// TIA Portal V19 export
TYPE "LEXCHANGETRAY_typeVfdProcessValues"
// simulated: Bool
// vfdStopped: Bool
// monitoring: LBC_typeSinaSpeedProcessValues
// stored: Access Published
   STRUCT
      simulated : Bool;
      vfdStopped : Bool;
      monitoring : "LBC_typeSinaSpeedProcessValues";
   END_STRUCT;
END_TYPE
